// TwinCAT 3 PLC project PlcProject
// ProgramVersion: 3.1.4023.0
// libraries:
//   Tc2_Standard, * (Beckhoff Automation GmbH)
//   Tc2_System, * (Beckhoff Automation GmbH)
//   Tc2_Utilities, * (Beckhoff Automation GmbH)
//   Tc3_Module, * (Beckhoff Automation GmbH)
// project tree:
//   GVLs/ GVL_HMI.TcGVL
//   / PlcTask.TcTTO
//   POUs/ FB_ChangeSystemTime.TcPOU, MAIN.TcPOU
// real-time tasks:
//   TASK PlcTask: cycle T#10ms, priority 20, ADS port 350

CONFIGURATION PlcProject
    RESOURCE PLC ON TwinCAT3
        TASK PlcTask(INTERVAL := T#10ms, PRIORITY := 20);
        PROGRAM MAIN WITH PlcTask : MAIN;
    END_RESOURCE
END_CONFIGURATION

// ---- GVLs/GVL_HMI.TcGVL
{attribute 'qualified_only'}
VAR_GLOBAL
	
	systemTime : TIMESTRUCT;
	
END_VAR

// ---- POUs/MAIN.TcPOU
PROGRAM MAIN
VAR
 fbChangeTime : FB_ChangeSystemTime;
END_VAR

fbChangeTime(systemTime:=GVL_Hmi.systemTime);

END_PROGRAM

// ---- POUs/FB_ChangeSystemTime.TcPOU
FUNCTION_BLOCK FB_ChangeSystemTime
VAR_INPUT
END_VAR
VAR_OUTPUT
	Error : BOOL;
	ErrorId : UDINT;
END_VAR
VAR_IN_OUT
	systemTime : TIMESTRUCT;
END_VAR
VAR
	enableWriteTime : BOOL;
	fbNtSetLocalTime : NT_SetLocalTime; 
	busyComplete : F_TRIG;
END_VAR

IF systemTime.wYear > 0 AND  systemTime.wMonth > 0 AND systemTime.wDay > 0 THEN 
	enableWriteTime := TRUE;
END_IF

fbNtSetLocalTime(START := (enableWriteTime AND NOT fbNtSetLocalTime.BUSY), TIMESTR := systemTime);
busyComplete(clk:= fbNtSetLocalTime.BUSY);

IF busyComplete.Q THEN
	enableWriteTime := FALSE;
	memset(ADR(systemTime),0,SIZEOF(systemTime));
	Error := fbNtSetLocalTime.ERR;
	ErrorId := fbNtSetLocalTime.ERRID;
END_IF

END_FUNCTION_BLOCK
